FUNCTION_BLOCK falhaFeedback (* Composite Function Block Type *)
  (* Standard: 61499-2 *)
  (* Version 0.0, 16/01/2026, Schneider Electric, template *)
  PACKAGE Hidryco.HidrycoLib;
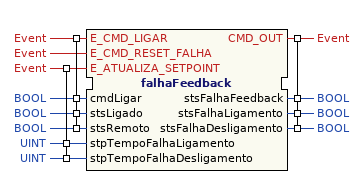
  EVENT_INPUT
    E_CMD_LIGAR WITH stsLigado, stsRemoto, cmdLigar;
    E_CMD_RESET_FALHA;
    E_ATUALIZA_SETPOINT WITH stpTempoFalhaLigamento, stpTempoFalhaDesligamento;
  END_EVENT
  EVENT_OUTPUT
    CMD_OUT WITH stsFalhaFeedback, stsFalhaLigamento, stsFalhaDesligamento;
  END_EVENT
  VAR_INPUT
    cmdLigar : BOOL;
    stsLigado : BOOL;
    stsRemoto : BOOL;
    stpTempoFalhaLigamento : UINT;
    stpTempoFalhaDesligamento : UINT;
  END_VAR
  VAR_OUTPUT
    stsFalhaFeedback : BOOL;
    stsFalhaLigamento : BOOL;
    stsFalhaDesligamento : BOOL;
  END_VAR
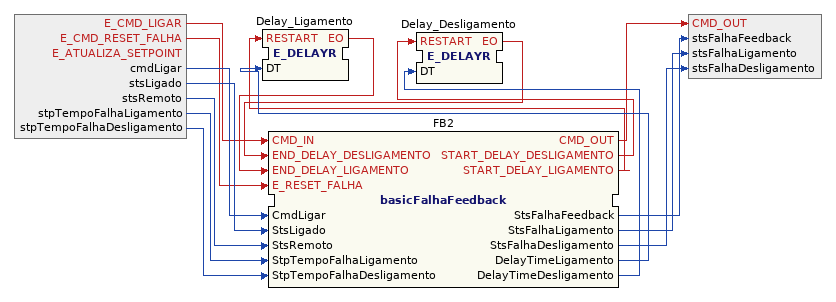
  FBS
    Delay_Ligamento : E_DELAYR;
    FB2 : basicFalhaFeedback;
    Delay_Desligamento : E_DELAYR;
  END_FBS
  EVENT_CONNECTIONS
    FB2.START_DELAY_DESLIGAMENTO TO Delay_Desligamento.RESTART;
    Delay_Desligamento.EO TO FB2.END_DELAY_DESLIGAMENTO;
    Delay_Ligamento.EO TO FB2.END_DELAY_LIGAMENTO;
    E_CMD_LIGAR TO FB2.CMD_IN;
    FB2.CMD_OUT TO CMD_OUT;
    E_CMD_RESET_FALHA TO FB2.E_RESET_FALHA;
    FB2.START_DELAY_LIGAMENTO TO Delay_Ligamento.RESTART;
  END_CONNECTIONS
  DATA_CONNECTIONS
    FB2.DelayTimeDesligamento TO Delay_Desligamento.DT;
    FB2.DelayTimeLigamento TO Delay_Ligamento.DT;
    stpTempoFalhaDesligamento TO FB2.StpTempoFalhaDesligamento;
    stpTempoFalhaLigamento TO FB2.StpTempoFalhaLigamento;
    stsRemoto TO FB2.StsRemoto;
    stsLigado TO FB2.StsLigado;
    cmdLigar TO FB2.CmdLigar;
    FB2.StsFalhaFeedback TO stsFalhaFeedback;
    FB2.StsFalhaLigamento TO stsFalhaLigamento;
    FB2.StsFalhaDesligamento TO stsFalhaDesligamento;
  END_CONNECTIONS
END_FUNCTION_BLOCK
